INTERFACE I_BYTE EXTENDS I_Datatype

{warning disable C5410}
PROPERTY PUBLIC Value : REFERENCE TO BYTE
{warning restore C5410}
GET
END_GET
END_PROPERTY

END_INTERFACE

(* stored: Version 1.1.0.1, ProductVersion 3.1.4024.15
   Itf I_BYTE: Id {77a835e4-1e75-06b5-2835-b3bd0416c447}
   Property Value: Id {9fcdef15-1b14-03fd-0931-94c86699178b}
   Get Get: Id {6368a136-8060-0f3e-12fd-9fc8d73afefc} *)
